PROGRAM PLC_TASK
VAR
END_VAR

END_PROGRAM

(* stored: Version 1.1.0.1, ProductVersion 3.1.4024.12
   POU PLC_TASK: Id {f6afb042-6086-4df6-8c54-dfc24e318219}, SpecialFunc None *)
